# EPICS substitutions: hugo/source/db/Beckhoff_3XXX/ecmcEL3702.substitutions
file "ecmc_analogInputArray-chX.template"
{
  pattern {CH_ID, DTYP,                FTVL    }
          {01,    "asynInt16ArrayIn",  "SHORT" }
          {02,    "asynInt16ArrayIn",  "SHORT" }
}

file "ecmcEL37XX-chX.template"
{
  pattern {CH_ID }
          {01    }
          {02    }
}

file "ecmcEL37XX_common.template"
{
  pattern {}
          {}
}
